PROGRAM HPP_HMI
VAR
	
	bTrig_SetptP					: BOOL;
	bTrig_SetptQ					: BOOL;
	bTrig_TargetSoCSoC				: BOOL;
	bTrig_TargetSoCP				: BOOL;
	bTrig_FreqRegParam				: BOOL;
	bTrig_UregParam					: BOOL;

	
	SetptP_IO						: REAL;
	SetptQ_IO						: REAL;
	                            	
	CalHppData						: PP;
	KK 								: UINT;
END_VAR

END_PROGRAM

(* stored: Version 1.1.0.1, ProductVersion 3.1.4024.12
   POU HPP_HMI: Id {a93e9070-7611-4686-acb3-183de167836c}, SpecialFunc None *)
